# EPICS StreamDevice protocol: ioc-tmo-output-couplerApp/tmo_couplerSup/devtmo_coupler.proto
Terminator = LF;

set_trim {
    out "trim \$1 \$2 \$3";
    in "%s";
}

set_switch {
    out "switch \$1 \$2";
    in "%s";
}

get_status {
    out "status \%1";
    in "Status Channel %*i = %X";
}

get_version {
    out "version";
    in "A=%s";
    in "B=%(\$1)s";
}
